// TIA Portal project "Paketband_mit_Hoehe_0" (V20)

(* hardware
DEVICE "S7-1500/ET200MP-Station_1"  S7-1500 station
   slot 0: "Profilschiene_0"  Rack  6ES7 590-1***0-0AA0
   slot 1: "PLC_1"  CPU 1513-1 PN  6ES7 513-1AM03-0AB0  V4.0
      slot 3: "CPU-Display_1"  6ES7591-1AA00-0AA0
      slot 32768: "PROFINET-Schnittstelle_1"  X1
         slot 32769: "Port_1"  X1 P1
         slot 32770: "Port_2"  X1 P2
      slot 34817: "Virtual CP interface port_1"  Virtual CP interface port  Virtual CP interface port FW V4.0
   slot 2: "DI 16x24VDC BA_1"  DI 16x24VDC BA  6ES7 521-1BH10-0AA0  V1.1
   slot 3: "DQ 16x24VDC/0.5A ST_1"  DQ 16x24VDC/0.5A ST  6ES7 522-1BH00-0AB0  V2.0
   slot 4: "AI 8xU/I/R/RTD BA_1"  AI 8xU/I/R/RTD BA  6ES7 531-7QF00-0AB0  V1.0
   slot 5: "AQ 8xU/I HS_1"  AQ 8xU/I HS  6ES7 532-5HF00-0AB0  V2.2
   slot 6: "AI 8xU/I/R/RTD BA_2"  AI 8xU/I/R/RTD BA  6ES7 531-7QF00-0AB0  V1.0
   slot 7: "AQ 8xU/I HS_2"  AQ 8xU/I HS  6ES7 532-5HF00-0AB0  V2.2
*)

// ===== PLC "PLC_1"  CPU 1513-1 PN =====

VAR_GLOBAL   // PLC tag table "Standard-Variablentabelle"
   "PlcLabConnectIn01" AT %ID32760 : DWord;
   "PlcLabConnectIn02" AT %ID32764 : DWord;
   "PlcLabConnectOut01" AT %QD32760 : DWord;
   "PlcLabConnectOut02" AT %QD32764 : DWord;
   "Anlage_aktiv" AT %M1.0 : Bool;
   "Clock_Byte" AT %MB0 : Byte;
   "Clock_10Hz" AT %M0.0 : Bool;
   "Clock_5Hz" AT %M0.1 : Bool;
   "Clock_2.5Hz" AT %M0.2 : Bool;
   "Clock_2Hz" AT %M0.3 : Bool;
   "Clock_1.25Hz" AT %M0.4 : Bool;
   "Clock_1Hz" AT %M0.5 : Bool;
   "Clock_0.625Hz" AT %M0.6 : Bool;
   "Clock_0.5Hz" AT %M0.7 : Bool;
   "Kleines_Paket" AT %M1.1 : Bool;
   "Mittleres_Paket" AT %M1.2 : Bool;
   "Großes_Paket" AT %M1.3 : Bool;
   "Betriebsstunden" AT %M20.0 : LTime;
   "Zaehler_kleine_Pakete" AT %MD30 : DInt;
   "Zaehler_mittlere_Pakete" AT %MD34 : DInt;
   "Zaehler_große_Pakete" AT %MD38 : DInt;
END_VAR

VAR_GLOBAL   // PLC tag table "Ausgaenge"
   "M1" AT %Q0.0 : Bool;   // Motor Förderband
   "H1" AT %Q0.1 : Bool;   // Meldeleuchte grün (Kleines Paket)
   "H2" AT %Q0.2 : Bool;   // Meldeleuchte gelb (Mittleres Paket)
   "H3" AT %Q0.3 : Bool;   // Meldeleuchte rot (Großes Paket)
   "H4" AT %Q0.4 : Bool;   // Leuchte Starttaster
   "H5" AT %Q0.5 : Bool;   // Leuchte Stopptaster
   "D1" AT %QD30 : DInt;   // Zähler (Kleine Pakete)
   "D2" AT %QD34 : DInt;   // Zähler (Mittlere Pakete)
   "D3" AT %QD38 : DInt;   // Zähler (Große Pakete)
   "D4" AT %QD42 : DInt;   // Gesamtzähler
END_VAR

VAR_GLOBAL   // PLC tag table "Eingaenge"
   "S1" AT %I0.0 : Bool;   // Starttaster
   "S2" AT %I0.1 : Bool;   // Stopptaster
   "1b1" AT %I0.2 : Bool;   // Sensor (Kleine Pakete)
   "1b2" AT %I0.3 : Bool;   // Sensor (Mittlere Pakete)
   "1b3" AT %I0.4 : Bool;   // Sensor (Große Pakete)
END_VAR

// folder: System blocks/Program resources

DATA_BLOCK "IEC_Timer_0_DB_1"   // DB1
{ S7_Optimized_Access := 'TRUE' }
AUTHOR : Simatic
FAMILY : IEC
NAME : IEC_LTMR
VERSION : 1.0
// stored: InstanceOfName IEC_LTIMER
"IEC_LTIMER"
BEGIN
END_DATA_BLOCK

// folder: (top level)

FUNCTION "Bandsteuerung" : Void   // FC1, FBD
{ S7_Optimized_Access := 'TRUE' }
VERSION : 0.1
   VAR_TEMP   // added for the SCL form of the ladder/FBD networks
      _w1 : Bool;
      _w2 : Bool;
   END_VAR
BEGIN

REGION Network 1: Förderbandsteuerung
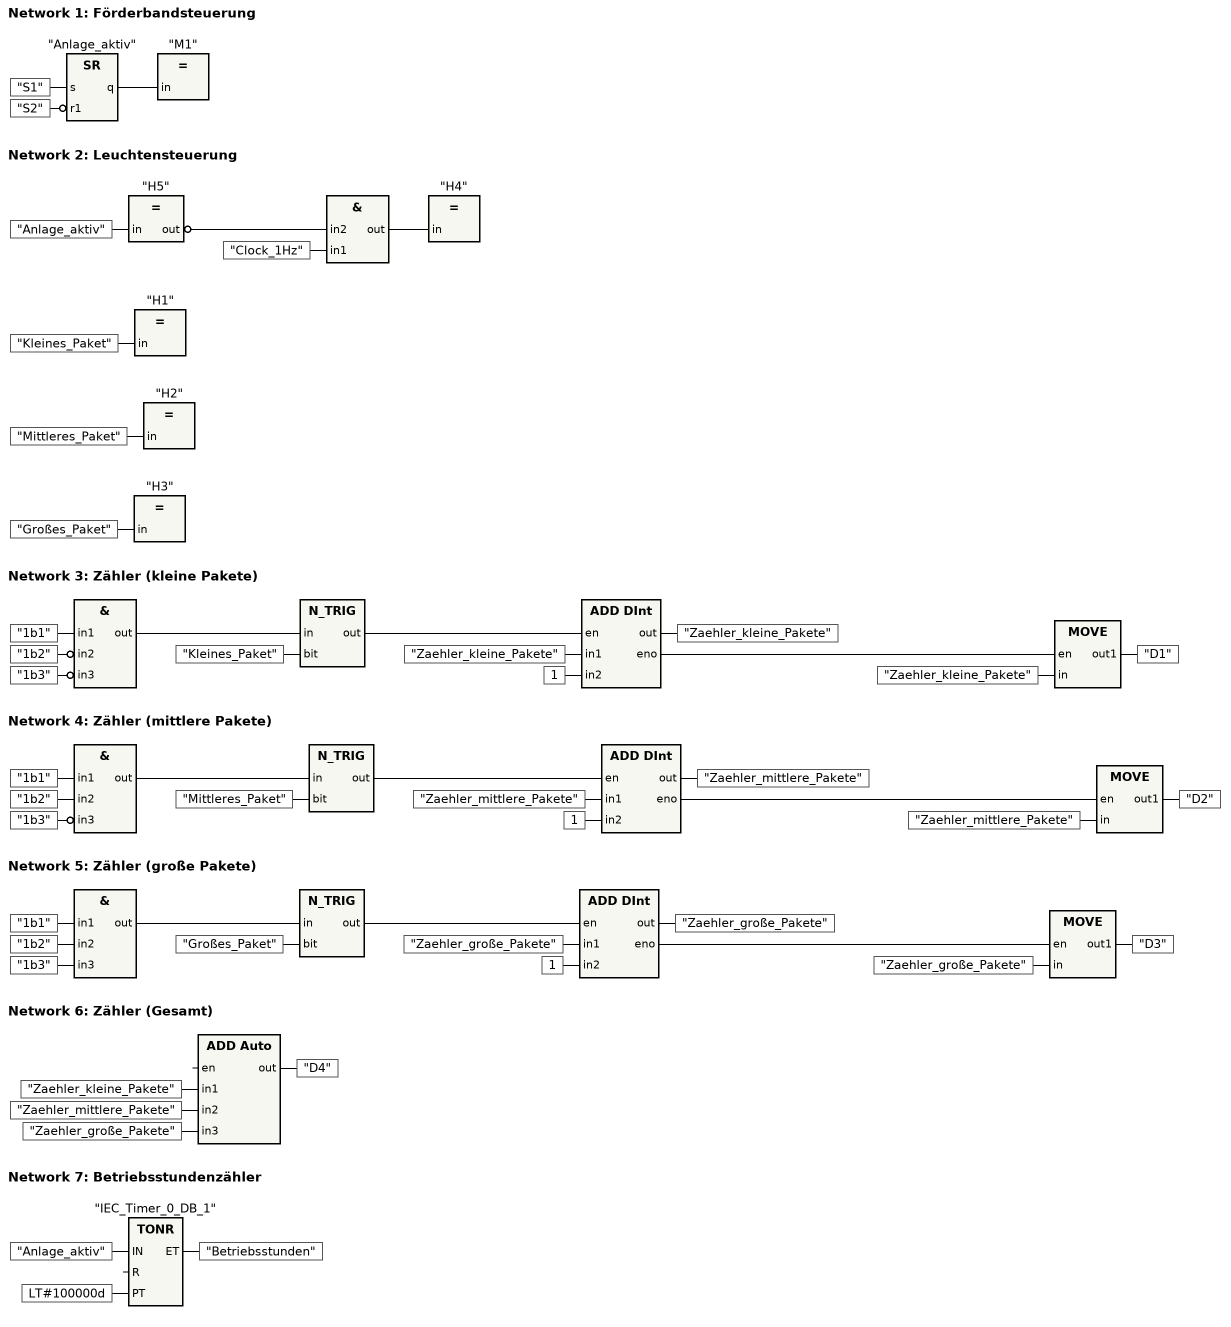
   IF "S1" THEN
       "Anlage_aktiv" := TRUE;   // SR flip-flop
   END_IF;
   IF NOT "S2" THEN "Anlage_aktiv" := FALSE; END_IF;
   "M1" := "Anlage_aktiv";
END_REGION

REGION Network 2: Leuchtensteuerung
   "H5" := "Anlage_aktiv";
   "H4" := NOT "Anlage_aktiv" AND "Clock_1Hz";
   "H1" := "Kleines_Paket";
   "H2" := "Mittleres_Paket";
   "H3" := "Großes_Paket";
END_REGION

REGION Network 3: Zähler (kleine Pakete)
   #_w1 := "1b1" AND NOT "1b2" AND NOT "1b3";
   #_w2 := NOT #_w1 AND "Kleines_Paket";   // falling edge
   "Kleines_Paket" := #_w1;
   IF #_w2 THEN
       "Zaehler_kleine_Pakete" := "Zaehler_kleine_Pakete" + 1;
       "D1" := "Zaehler_kleine_Pakete";
   END_IF;
END_REGION

REGION Network 4: Zähler (mittlere Pakete)
   #_w1 := "1b1" AND "1b2" AND NOT "1b3";
   #_w2 := NOT #_w1 AND "Mittleres_Paket";   // falling edge
   "Mittleres_Paket" := #_w1;
   IF #_w2 THEN
       "Zaehler_mittlere_Pakete" := "Zaehler_mittlere_Pakete" + 1;
       "D2" := "Zaehler_mittlere_Pakete";
   END_IF;
END_REGION

REGION Network 5: Zähler (große Pakete)
   #_w1 := "1b1" AND "1b2" AND "1b3";
   #_w2 := NOT #_w1 AND "Großes_Paket";   // falling edge
   "Großes_Paket" := #_w1;
   IF #_w2 THEN
       "Zaehler_große_Pakete" := "Zaehler_große_Pakete" + 1;
       "D3" := "Zaehler_große_Pakete";
   END_IF;
END_REGION

REGION Network 6: Zähler (Gesamt)
   "D4" := "Zaehler_kleine_Pakete" + "Zaehler_mittlere_Pakete" + "Zaehler_große_Pakete";
END_REGION

REGION Network 7: Betriebsstundenzähler
   "IEC_Timer_0_DB_1".TONR(IN := "Anlage_aktiv", PT := LT#100000d, ET => "Betriebsstunden");
END_REGION
END_FUNCTION

ORGANIZATION_BLOCK "Main"   // OB1, FBD, ProgramCycle
TITLE = "Main Program Sweep (Cycle)"
{ S7_Optimized_Access := 'TRUE' }
VERSION : 0.1
   VAR_INPUT
      Initial_Call : Bool;   // Initial call of this OB
      Remanence : Bool;   // =True, if remanent data are available
   END_VAR
BEGIN

REGION Network 1
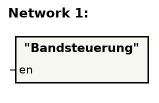
   "Bandsteuerung"();
END_REGION
END_ORGANIZATION_BLOCK